(* Logix 5000 project; controller GP1 vendor 1 type 14 code 155 rev 32.11; software revision 32.01 *)
// GP1

TASK MainTask (continuous, watchdog 500 ms) : MainProgram

MODULES
   Local : vendor 1 type 14 code 155 (PointIO 0, rev 32.11)
      GP1_INPUT_MODULE_4 : 1734-IB8 (PointIO 4, rev 3.1, Input RPI 20 ms)
           Local:4:I.Data.0   // FC TOPE
           Local:4:I.Data.1   // IC TOPE
           Local:4:I.Data.3   // CAPACITIVO IZQUIERDO
           Local:4:I.Data.6   // CAPACITIVO DERECHO
      GP1_INPUT_MODULE_5 : 1734-IB8 (PointIO 5, rev 3.1, Input RPI 20 ms)
           Local:5:I.Data.0   // INDUCTIVO TOPE
           Local:5:I.Data.2   // ARRANQUE
           Local:5:I.Data.1   // PARO
           Local:5:I.Data.3   // BOTON REARME
      GP1_OUTPUT_MODULE_3 : 1734-OB8 (PointIO 3, rev 3.1, Output RPI 20 ms)
      GP1_OUTPUT_MODULE_2 : 1734-OB8 (PointIO 2, rev 3.1, Output RPI 20 ms)
           Local:2:O.Data.0   // YELLOW
           Local:2:O.Data.1   // RED
           Local:2:O.Data.2   // AZUL
      Discrete_IO : Embedded (PointIO 1, rev 32.11, Output RPI 20 ms)
           Local:1:I.Data.12   // FC CORTE SUPERIOR
           Local:1:I.Data.6   // FC CLAMP VERTICAL
           Local:1:I.Data.10   // IC CLAMP
           Local:1:I.Data.11   // FC CLAMP
           Local:1:I.Data.2   // IC NAVAJAS 3 L
           Local:1:I.Data.7   // IC CLAMP VERTICAL
           Local:1:I.Data.0   // FC NAVAJA 1
           Local:1:I.Data.1   // IC NAVAJA 1
           Local:1:I.Data.3   // FC NAVAJAS 3 L
           Local:1:I.Data.13   // IC CORTE SUPERIOR
           Local:1:I.Data.8   // IC NAVAJAS 3 R
           Local:1:I.Data.14   // IC TROQUEL
           Local:1:I.Data.15   // FC TROQUEL
           Local:1:I.Data.9   // FC NAVAJAS 3 R
           Local:1:I.Data.4   // FC CLAMP HORIZONTAL
           Local:1:I.Data.5   // IC CLAMP HORIZONTAL
           Local:1:O.Data.15   // GREEN
END_MODULES

VAR_GLOBAL   (* controller tags *)
   ACT0_OFF : BOOL := 1;   // NAVAJAS 3 R OFF
   ACT0_ON : BOOL;   // NAVAJAS 3 R ON
   ACT1_OFF : BOOL := 1;   // TROQUEL OFF
   ACT1_ON : BOOL;   // TROQUEL ON
   ACT2_OFF : BOOL := 1;   // CORTE SUPERIOR OFF
   ACT2_ON : BOOL;   // CORTE SUPERIOR ON
   ACT3_OFF : BOOL := 1;   // NAVAJA 1 OFF
   ACT3_ON : BOOL;   // NAVAJA 1 ON
   ACT4_OFF : BOOL;   // CLAMP VERTICAL OFF
   ACT4_ON : BOOL := 1;   // CLAMP VERTICAL ON
   ACT5_OFF : BOOL := 1;   // CLAMP OFF
   ACT5_ON : BOOL;   // CLAMP ON
   ACT6_OFF : BOOL;   // CLAMP HORIZONTAL OFF
   ACT6_ON : BOOL := 1;   // CLAMP HORIZONTAL ON
   ACT7_OFF : BOOL := 1;   // NAVAJA 3 L OFF
   ACT7_ON : BOOL;   // NAVAJA 3 L ON
   ACT8_OFF : BOOL;   // TOPE OFF
   ACT8_ON : BOOL := 1;   // TOPE ON
   AIR_ALARM : BOOL;
   ALARM_TIM : TIMER := (PRE := 5000);
   ALARMED : BOOL;
   ARRANQUE_AUTO : BOOL;
   AUTO : BOOL;
   C1 : COUNTER := (ACC := 5, DN := 1);
   CAPACITIVE_SENSOR_1 : BOOL;
   CAPACITIVE_SENSOR_2 : BOOL;
   CND1 : BOOL;
   CND10 : BOOL;
   CND2 : BOOL;
   CND3 : BOOL;
   CND4 : BOOL;
   CND5 : BOOL;
   CND6 : BOOL;
   CND7 : BOOL;
   CND8 : BOOL;
   CND9 : BOOL;
   CORTE_VALVULA : BOOL;
   CORTINA_SEG : BOOL := 1;
   CT : COUNTER := (ACC := 47, DN := 1);
   CURRENT_SCREEN : DINT;
   E_STOP : BOOL;
   E_STOP_ALARM : BOOL;
   EstadoHMI : DINT := 2;
   EVBI0_AUTO_OFF : BOOL;   // NAVAJAS 3 OFF AUTO
   EVBI0_AUTO_ON : BOOL;   // NAVAJAS 3 ON AUTO
   EVBI0_MAN_OFF : BOOL;   // NAVAJAS 3 OFF MANUAL
   EVBI0_MAN_ON : BOOL;   // NAVAJAS 3 ON MANUAL
   EVBI0_OFF : BOOL := 1;   // NAVAJAS 3 OFF
   EVBI0_ON : BOOL;   // NAVAJAS 3 ON
   EVBI1_AUTO_OFF : BOOL;   // TROQUEL OFF AUTO
   EVBI1_AUTO_ON : BOOL;   // TROQUEL ON AUTO
   EVBI1_MAN_OFF : BOOL;   // TROQUEL OFF MANUAL
   EVBI1_MAN_ON : BOOL;   // TROQUEL ON MANUAL
   EVBI1_OFF : BOOL := 1;   // TROQUEL OFF
   EVBI1_ON : BOOL;   // TROQUEL ON
   EVBI2_AUTO_OFF : BOOL;   // CLAMP OFF AUTO
   EVBI2_AUTO_ON : BOOL;   // CLAMP ON AUTO
   EVBI2_MAN_OFF : BOOL;   // CLAMP OFF MANUAL
   EVBI2_MAN_ON : BOOL;   // CLAMP ON MANUAL
   EVBI2_OFF : BOOL := 1;   // CLAMP OFF
   EVBI2_ON : BOOL;   // CLAMP ON
   EVBI3_AUTO_OFF : BOOL;   // NAVAJA 1 OFF AUTO
   EVBI3_AUTO_ON : BOOL;   // NAVAJA 1 ON AUTO
   EVBI3_MAN_OFF : BOOL;   // NAVAJA 1 OFF MANUAL
   EVBI3_MAN_ON : BOOL;   // NAVAJA 1 ON MANUAL
   EVBI3_OFF : BOOL := 1;   // NAVAJA 1 OFF
   EVBI3_ON : BOOL;   // NAVAJA 1 ON
   EVBI4_AUTO_OFF : BOOL;   // CLAMP VERTICAL OFF AUTO
   EVBI4_AUTO_ON : BOOL;   // CLAMP VERTICAL ON AUTO
   EVBI4_MAN_OFF : BOOL;   // CLAMP VERTICAL OFF MANUAL
   EVBI4_MAN_ON : BOOL;   // CLAMP VERTICAL ON MANUAL
   EVBI4_OFF : BOOL;   // CLAMP VERTICAL OFF
   EVBI4_ON : BOOL := 1;   // CLAMP VERTICAL ON
   EVBI5_AUTO_OFF : BOOL;   // CORTE SUPERIOR OFF AUTO
   EVBI5_AUTO_ON : BOOL;   // CORTE SUPERIOR ON AUTO
   EVBI5_MAN_OFF : BOOL;   // CORTE SUPERIOR OFF MANUAL
   EVBI5_MAN_ON : BOOL;   // CORTE SUPERIOR ON MANUAL
   EVBI5_OFF : BOOL := 1;   // CORTE SUPERIOR OFF
   EVBI5_ON : BOOL;   // CORTE SUPERIOR ON
   EVBI6_AUTO_OFF : BOOL;   // CLAMP HORIZONTAL OFF AUTO
   EVBI6_AUTO_ON : BOOL;   // CLAMP HORIZONTAL ON AUTO
   EVBI6_MAN_OFF : BOOL;   // CLAMP HORIZONTAL OFF MANUAL
   EVBI6_MAN_ON : BOOL;   // CLAMP HORIZONTAL ON MANUAL
   EVBI6_OFF : BOOL;   // CLAMP HORIZONTAL OFF
   EVBI6_ON : BOOL := 1;   // CLAMP HORIZONTAL ON
   EVMONO1_AUTO_OFF : BOOL;
   EVMONO1_AUTO_ON : BOOL;   // TOPE_AUTO_ON
   EVMONO1_MAN_OFF : BOOL;
   EVMONO1_MAN_ON : BOOL;
   EVMONO_OFF : BOOL;
   EVMONO_ON : BOOL;   // TOPE ON
   EXCEDDED_TIME_FOR_CILINDERS : BOOL;
   EXCEDDED_TIME_FOR_INIT_COND : BOOL;
   FAIL_COUNT : COUNTER;
   GREEN_LIGHT : BOOL;
   INITIAL_CONDITIONS_NOT_READY : BOOL := 1;
   INITIAL_CONDITIONS_READY : BOOL;
   L_S_OK : BOOL := 1;   // SENSOR IZQUIERDO
   LAMP : BOOL := 1;
   LATCH_TEST : BOOL;
   LIGHT_CURTAIN : BOOL;
   MAN_SCREENS : BOOL;   // PANTALLAS MANUALES
   MANUAL : BOOL := 1;
   MSJ_CND_INIT : DINT := 8;
   NO_AIR : BOOL;
   NO_ALARM : BOOL := 1;
   NOT_CORRECTLY_PLACED : BOOL;
   OBESTOP : BOOL;
   OK : BOOL;
   ONS1 : BOOL;
   PARO : BOOL := 1;
   Paso1 : BOOL;
   Paso10 : BOOL;
   Paso11 : BOOL;
   Paso12 : BOOL;
   Paso13 : BOOL;
   Paso14 : BOOL;
   Paso15 : BOOL;
   Paso16 : BOOL;
   Paso17 : BOOL;
   Paso18 : BOOL;
   Paso2 : BOOL;
   Paso3 : BOOL;
   Paso4 : BOOL;
   Paso5 : BOOL;
   Paso6 : BOOL;
   Paso7 : BOOL;
   Paso8 : BOOL;
   Paso9 : BOOL;
   Paso_Sec : DINT;
   PIECE_PLACED : BOOL;
   PRESOSTATO : BOOL := 1;
   R_S_OK : BOOL := 1;   // SENSOR DERECHO
   REARME_OK : BOOL;
   REARMY_BUTTON : BOOL;
   REARMY_TIME : TIMER := (PRE := 5);
   REARMY_WARNING : BOOL := 1;   // LUZ DE ARME
   RED_LIGHT : BOOL;
   REPEATED_ALARM : BOOL;
   RESET_COUNTER : BOOL;
   RESET_LATCH_TEST : BOOL;
   SAFETY_CURTAIN : BOOL;
   SAFETY_CURTAIN_ALARM : BOOL;
   SBESTOP : BOOL;
   SENSOR1 : BOOL;
   SENSOR_TOPE : BOOL;   // TOPE DE PIEZA
   Sequence_ON : BOOL;
   Start_Sequence : BOOL;
   T1 : TIMER := (PRE := 300);
   T10 : TIMER := (PRE := 300);
   T11 : TIMER := (PRE := 300);
   T12 : TIMER := (PRE := 300);
   T13 : TIMER := (PRE := 300);
   T14 : TIMER := (PRE := 300);
   T15 : TIMER := (PRE := 300);
   T16 : TIMER := (PRE := 300);
   T17 : TIMER := (PRE := 300);
   T18 : TIMER := (PRE := 1000);
   T2 : TIMER := (PRE := 300);
   T3 : TIMER := (PRE := 300);
   T4 : TIMER := (PRE := 300);
   T5 : TIMER := (PRE := 300);
   T6 : TIMER := (PRE := 300);
   T7 : TIMER := (PRE := 300);
   T8 : TIMER := (PRE := 300);
   T9 : TIMER := (PRE := 300);
   TCLAMP : TIMER := (PRE := 250, ACC := 250, EN := 1, DN := 1);
   TEST : BOOL;
   TEST_2 : BOOL;
   TEST_3 : BOOL;
   TEST_RESET : BOOL;
   TEST_STOP : BOOL;
   TIMOFF : TIMER := (PRE := 500);
   TIMON : TIMER := (PRE := 500);
   TIMSACC : DINT;
   TIMW1 : TIMER := (PRE := 2000);
   TIMW2 : TIMER := (PRE := 1);
   USER : DINT;
   WAITING : BOOL;
   WORKING : BOOL;
   YELLOW_LIGHT : BOOL := 1;
END_VAR

PROGRAM MainProgram   (* main routine MainRoutine *)
VAR
   BYPASS_DER : BOOL;
   BYPASS_IZQ : BOOL;
   BYPASS_TOPE : BOOL;
   BypassStatus : DINT;
   CERRARSESION : BOOL;
   ING_ACCESS : BOOL;
   LOGOUT : BOOL;
   MTTO_ACCESS : BOOL;
   RESET_COUNTERT : BOOL;
   TEMP1 : BOOL;
   TEMP2 : BOOL;
   TEMP3 : BOOL;
   USERstring : STRING;
END_VAR

ROUTINE ALARMS   (* ladder *)
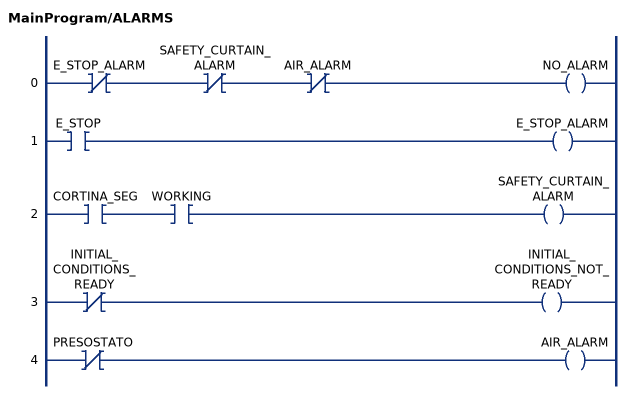
   0: XIO(E_STOP_ALARM)XIO(SAFETY_CURTAIN_ALARM)XIO(AIR_ALARM)OTE(NO_ALARM);
   1: XIC(E_STOP)OTE(E_STOP_ALARM);
   2: XIC(CORTINA_SEG)XIC(WORKING)OTE(SAFETY_CURTAIN_ALARM);
   3: XIO(INITIAL_CONDITIONS_READY)OTE(INITIAL_CONDITIONS_NOT_READY);
   4: XIO(PRESOSTATO)OTE(AIR_ALARM);
END_ROUTINE

ROUTINE AUTO_SEQUENCE   (* ladder *)
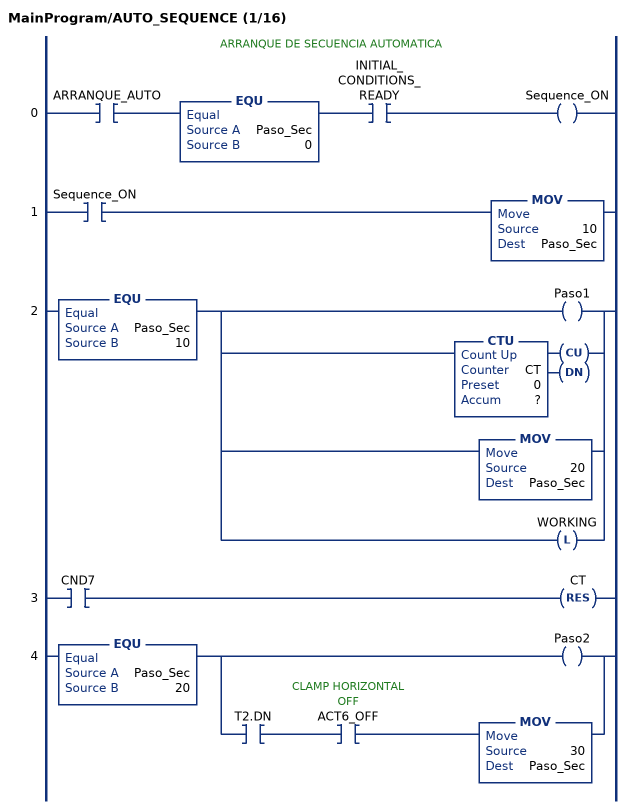
   // ARRANQUE DE SECUENCIA AUTOMATICA
   0: XIC(ARRANQUE_AUTO)EQU(Paso_Sec,0)XIC(INITIAL_CONDITIONS_READY)OTE(Sequence_ON);
   1: XIC(Sequence_ON)MOV(10,Paso_Sec);
   2: EQU(Paso_Sec,10)[OTE(Paso1) ,CTU(CT,?,?) ,MOV(20,Paso_Sec) ,OTL(WORKING) ];
   3: XIC(CND7)RES(CT);
   4: EQU(Paso_Sec,20)[OTE(Paso2) ,XIC(T2.DN) XIC(ACT6_OFF) MOV(30,Paso_Sec) ];
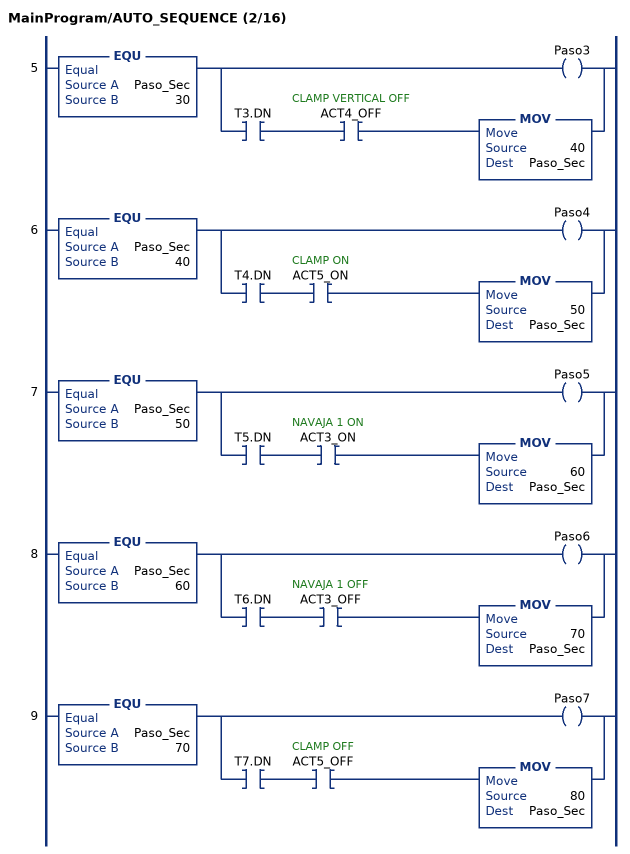
   5: EQU(Paso_Sec,30)[OTE(Paso3) ,XIC(T3.DN) XIC(ACT4_OFF) MOV(40,Paso_Sec) ];
   6: EQU(Paso_Sec,40)[OTE(Paso4) ,XIC(T4.DN) XIC(ACT5_ON) MOV(50,Paso_Sec) ];
   7: EQU(Paso_Sec,50)[OTE(Paso5) ,XIC(T5.DN) XIC(ACT3_ON) MOV(60,Paso_Sec) ];
   8: EQU(Paso_Sec,60)[OTE(Paso6) ,XIC(T6.DN) XIC(ACT3_OFF) MOV(70,Paso_Sec) ];
   9: EQU(Paso_Sec,70)[OTE(Paso7) ,XIC(T7.DN) XIC(ACT5_OFF) MOV(80,Paso_Sec) ];
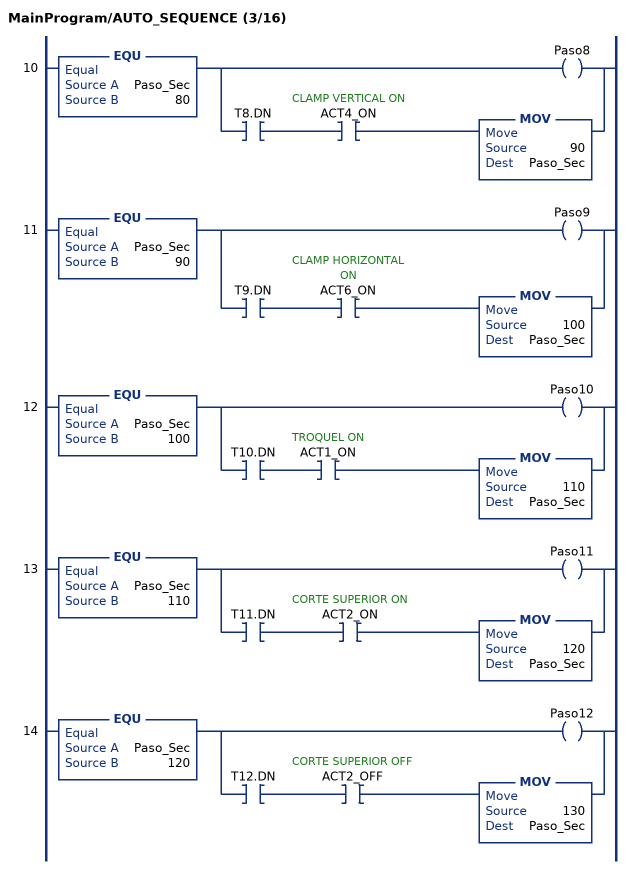
   10: EQU(Paso_Sec,80)[OTE(Paso8) ,XIC(T8.DN) XIC(ACT4_ON) MOV(90,Paso_Sec) ];
   11: EQU(Paso_Sec,90)[OTE(Paso9) ,XIC(T9.DN) XIC(ACT6_ON) MOV(100,Paso_Sec) ];
   12: EQU(Paso_Sec,100)[OTE(Paso10) ,XIC(T10.DN) XIC(ACT1_ON) MOV(110,Paso_Sec) ];
   13: EQU(Paso_Sec,110)[OTE(Paso11) ,XIC(T11.DN) XIC(ACT2_ON) MOV(120,Paso_Sec) ];
   14: EQU(Paso_Sec,120)[OTE(Paso12) ,XIC(T12.DN) XIC(ACT2_OFF) MOV(130,Paso_Sec) ];
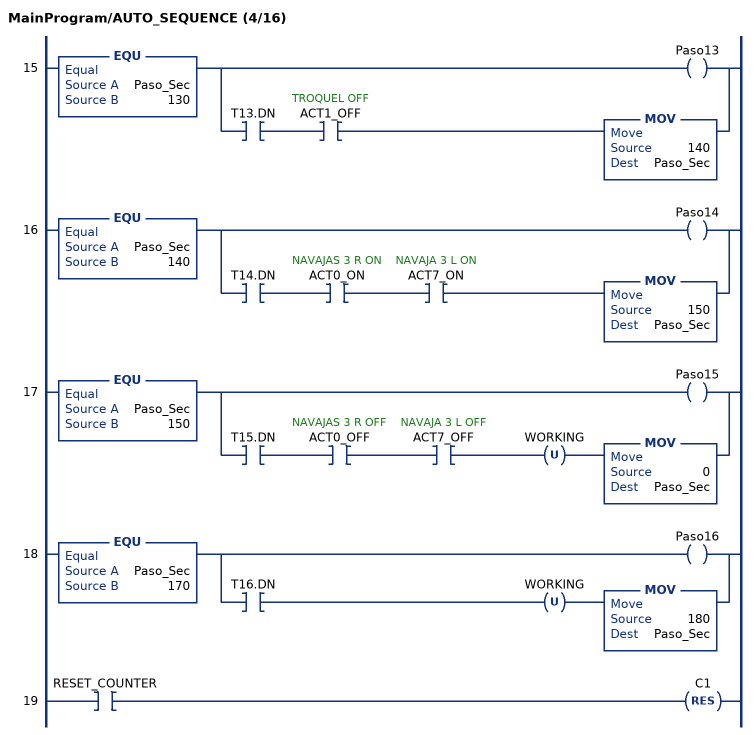
   15: EQU(Paso_Sec,130)[OTE(Paso13) ,XIC(T13.DN) XIC(ACT1_OFF) MOV(140,Paso_Sec) ];
   16: EQU(Paso_Sec,140)[OTE(Paso14) ,XIC(T14.DN) XIC(ACT0_ON) XIC(ACT7_ON) MOV(150,Paso_Sec) ];
   17: EQU(Paso_Sec,150)[OTE(Paso15) ,XIC(T15.DN) XIC(ACT0_OFF) XIC(ACT7_OFF) OTU(WORKING) MOV(0,Paso_Sec) ];
   18: EQU(Paso_Sec,170)[OTE(Paso16) ,XIC(T16.DN) OTU(WORKING) MOV(180,Paso_Sec) ];
   19: XIC(RESET_COUNTER)RES(C1);
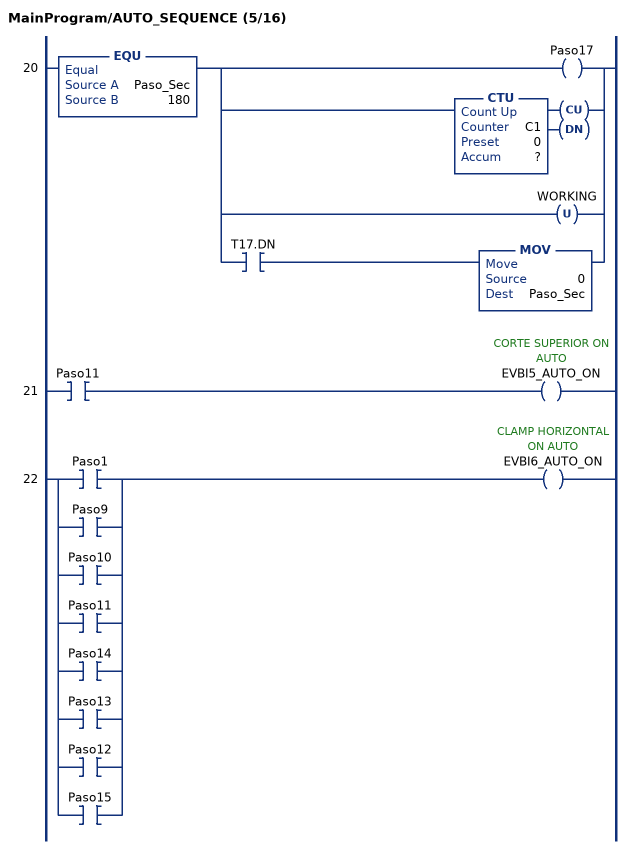
   20: EQU(Paso_Sec,180)[OTE(Paso17) ,CTU(C1,?,?) ,OTU(WORKING) ,XIC(T17.DN) MOV(0,Paso_Sec) ];
   21: XIC(Paso11)OTE(EVBI5_AUTO_ON);
   22: [XIC(Paso1) ,XIC(Paso9) ,XIC(Paso10) ,XIC(Paso11) ,XIC(Paso14) ,XIC(Paso13) ,XIC(Paso12) ,XIC(Paso15) ]OTE(EVBI6_AUTO_ON);
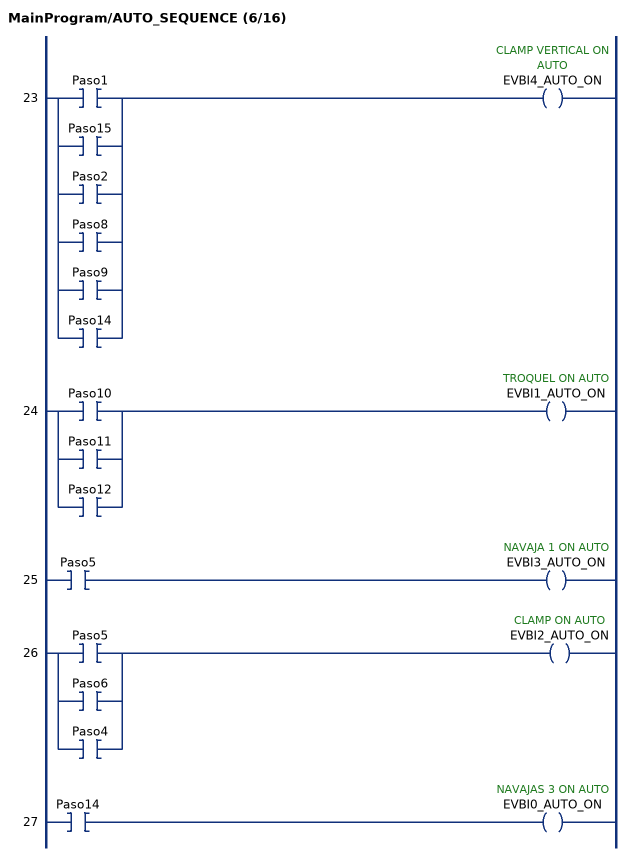
   23: [XIC(Paso1) ,XIC(Paso15) ,XIC(Paso2) ,XIC(Paso8) ,XIC(Paso9) ,XIC(Paso14) ]OTE(EVBI4_AUTO_ON);
   24: [XIC(Paso10) ,XIC(Paso11) ,XIC(Paso12) ]OTE(EVBI1_AUTO_ON);
   25: XIC(Paso5)OTE(EVBI3_AUTO_ON);
   26: [XIC(Paso5) ,XIC(Paso6) ,XIC(Paso4) ]OTE(EVBI2_AUTO_ON);
   27: XIC(Paso14)OTE(EVBI0_AUTO_ON);
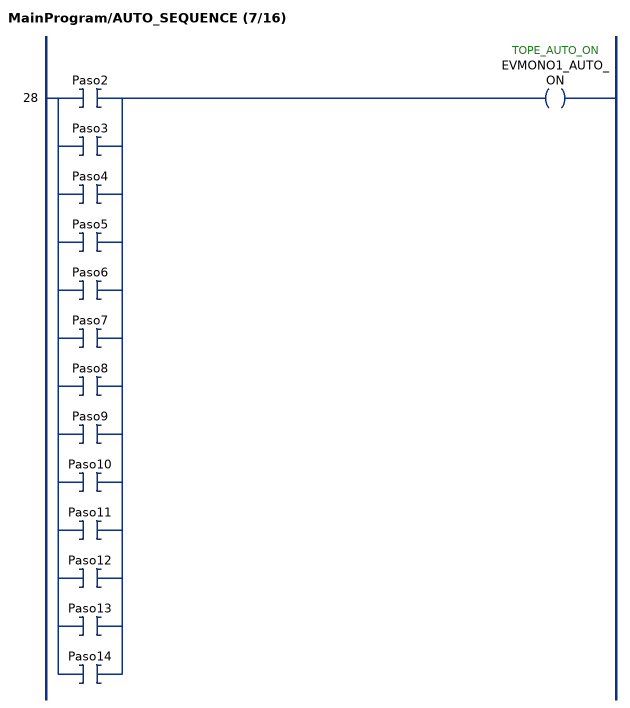
   28: [XIC(Paso2) ,XIC(Paso3) ,XIC(Paso4) ,XIC(Paso5) ,XIC(Paso6) ,XIC(Paso7) ,XIC(Paso8) ,XIC(Paso9) ,XIC(Paso10) ,XIC(Paso11) ,XIC(Paso12) ,XIC(Paso13) ,XIC(Paso14) ]OTE(EVMONO1_AUTO_ON);
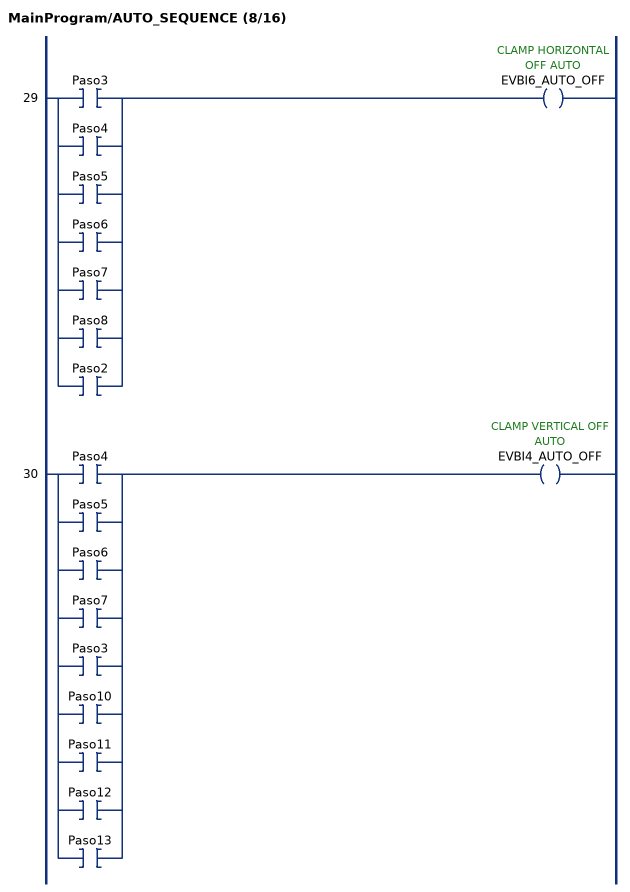
   29: [XIC(Paso3) ,XIC(Paso4) ,XIC(Paso5) ,XIC(Paso6) ,XIC(Paso7) ,XIC(Paso8) ,XIC(Paso2) ]OTE(EVBI6_AUTO_OFF);
   30: [XIC(Paso4) ,XIC(Paso5) ,XIC(Paso6) ,XIC(Paso7) ,XIC(Paso3) ,XIC(Paso10) ,XIC(Paso11) ,XIC(Paso12) ,XIC(Paso13) ]OTE(EVBI4_AUTO_OFF);
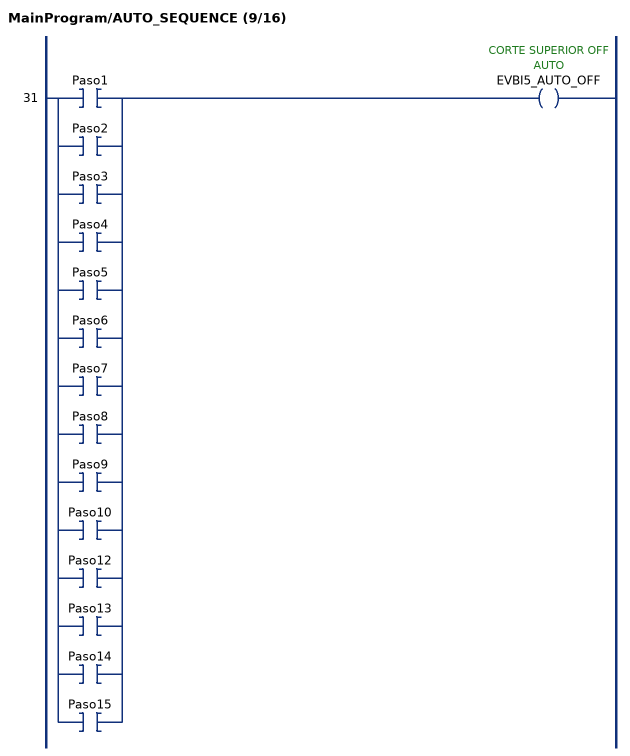
   31: [XIC(Paso1) ,XIC(Paso2) ,XIC(Paso3) ,XIC(Paso4) ,XIC(Paso5) ,XIC(Paso6) ,XIC(Paso7) ,XIC(Paso8) ,XIC(Paso9) ,XIC(Paso10) ,XIC(Paso12) ,XIC(Paso13) ,XIC(Paso14) ,XIC(Paso15) ]OTE(EVBI5_AUTO_OFF);
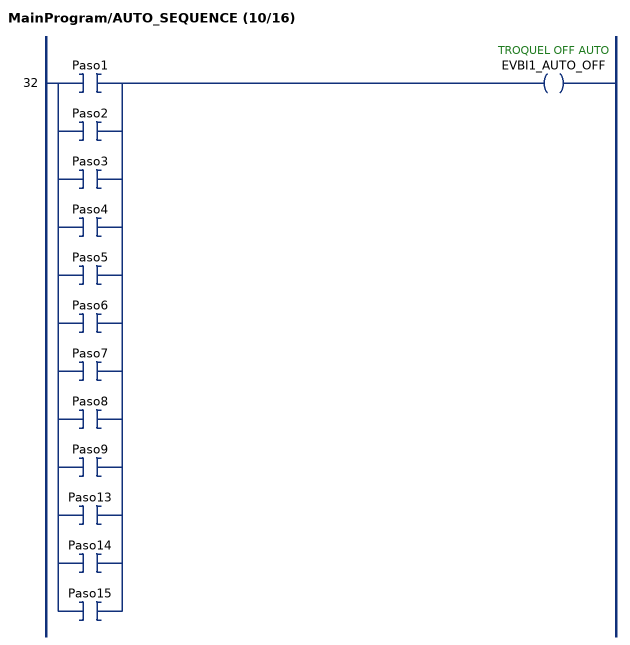
   32: [XIC(Paso1) ,XIC(Paso2) ,XIC(Paso3) ,XIC(Paso4) ,XIC(Paso5) ,XIC(Paso6) ,XIC(Paso7) ,XIC(Paso8) ,XIC(Paso9) ,XIC(Paso13) ,XIC(Paso14) ,XIC(Paso15) ]OTE(EVBI1_AUTO_OFF);
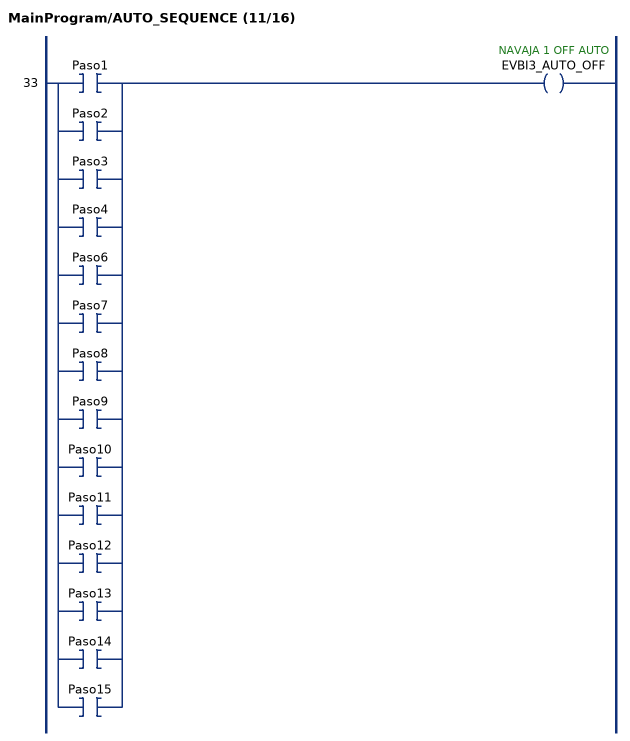
   33: [XIC(Paso1) ,XIC(Paso2) ,XIC(Paso3) ,XIC(Paso4) ,XIC(Paso6) ,XIC(Paso7) ,XIC(Paso8) ,XIC(Paso9) ,XIC(Paso10) ,XIC(Paso11) ,XIC(Paso12) ,XIC(Paso13) ,XIC(Paso14) ,XIC(Paso15) ]OTE(EVBI3_AUTO_OFF);
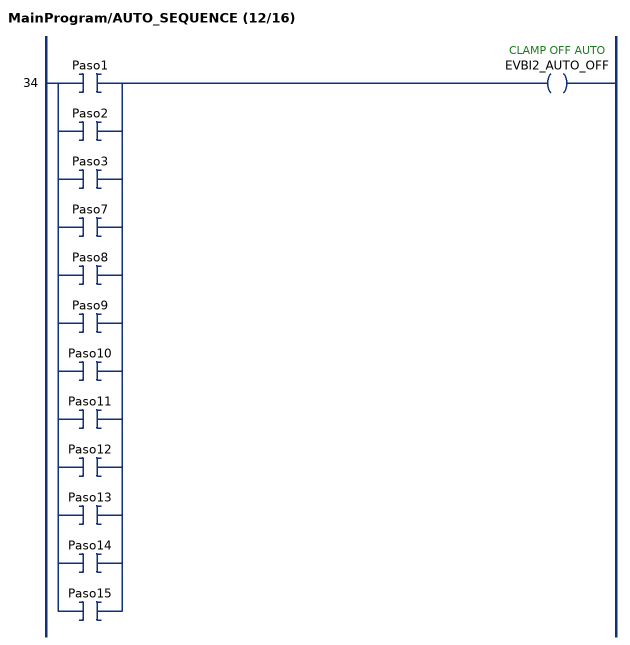
   34: [XIC(Paso1) ,XIC(Paso2) ,XIC(Paso3) ,XIC(Paso7) ,XIC(Paso8) ,XIC(Paso9) ,XIC(Paso10) ,XIC(Paso11) ,XIC(Paso12) ,XIC(Paso13) ,XIC(Paso14) ,XIC(Paso15) ]OTE(EVBI2_AUTO_OFF);
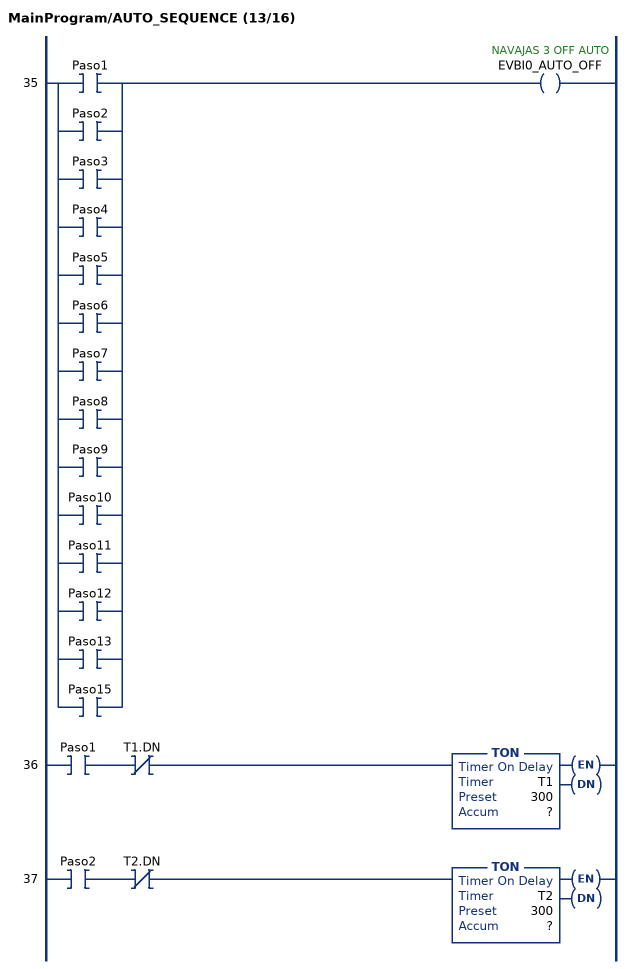
   35: [XIC(Paso1) ,XIC(Paso2) ,XIC(Paso3) ,XIC(Paso4) ,XIC(Paso5) ,XIC(Paso6) ,XIC(Paso7) ,XIC(Paso8) ,XIC(Paso9) ,XIC(Paso10) ,XIC(Paso11) ,XIC(Paso12) ,XIC(Paso13) ,XIC(Paso15) ]OTE(EVBI0_AUTO_OFF);
   36: XIC(Paso1)XIO(T1.DN)TON(T1,?,?);
   37: XIC(Paso2)XIO(T2.DN)TON(T2,?,?);
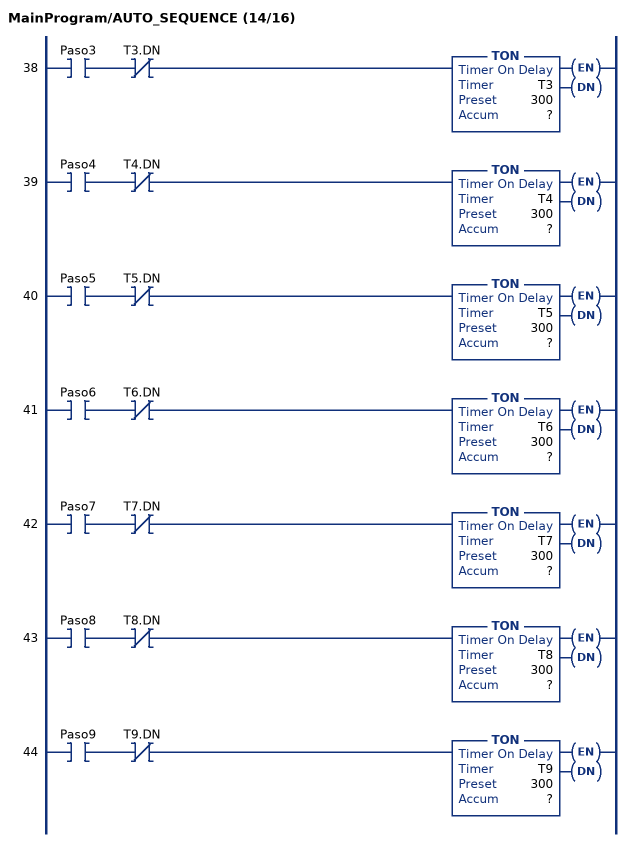
   38: XIC(Paso3)XIO(T3.DN)TON(T3,?,?);
   39: XIC(Paso4)XIO(T4.DN)TON(T4,?,?);
   40: XIC(Paso5)XIO(T5.DN)TON(T5,?,?);
   41: XIC(Paso6)XIO(T6.DN)TON(T6,?,?);
   42: XIC(Paso7)XIO(T7.DN)TON(T7,?,?);
   43: XIC(Paso8)XIO(T8.DN)TON(T8,?,?);
   44: XIC(Paso9)XIO(T9.DN)TON(T9,?,?);
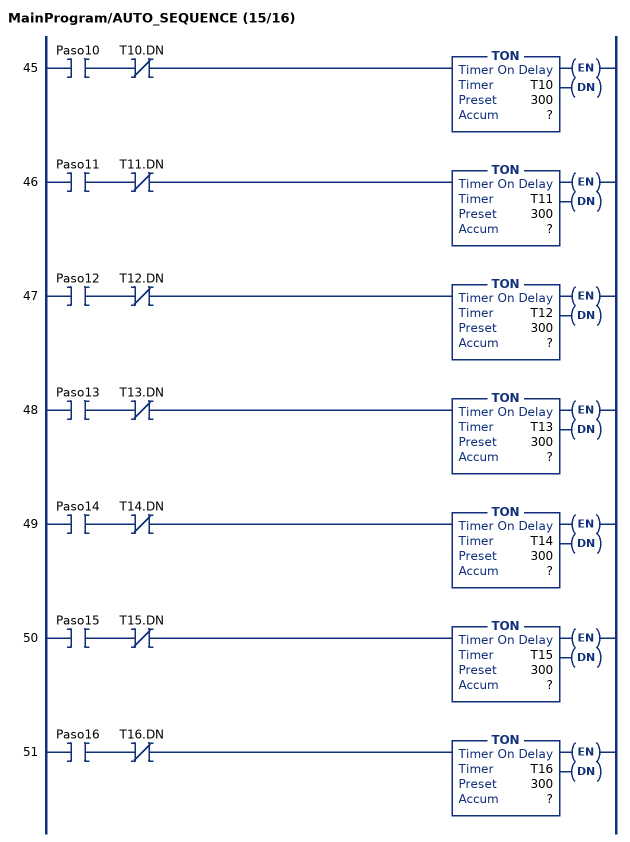
   45: XIC(Paso10)XIO(T10.DN)TON(T10,?,?);
   46: XIC(Paso11)XIO(T11.DN)TON(T11,?,?);
   47: XIC(Paso12)XIO(T12.DN)TON(T12,?,?);
   48: XIC(Paso13)XIO(T13.DN)TON(T13,?,?);
   49: XIC(Paso14)XIO(T14.DN)TON(T14,?,?);
   50: XIC(Paso15)XIO(T15.DN)TON(T15,?,?);
   51: XIC(Paso16)XIO(T16.DN)TON(T16,?,?);
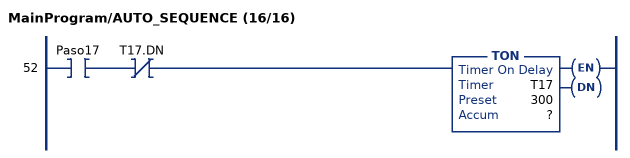
   52: XIC(Paso17)XIO(T17.DN)TON(T17,?,?);
END_ROUTINE

ROUTINE INPUTS   (* ladder *)
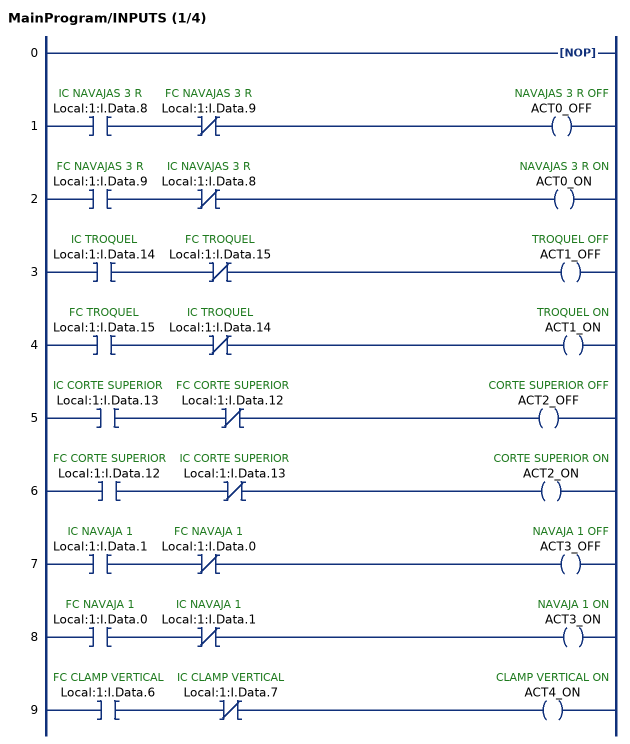
   0: NOP();
   1: XIC(Local:1:I.Data.8)XIO(Local:1:I.Data.9)OTE(ACT0_OFF);
   2: XIC(Local:1:I.Data.9)XIO(Local:1:I.Data.8)OTE(ACT0_ON);
   3: XIC(Local:1:I.Data.14)XIO(Local:1:I.Data.15)OTE(ACT1_OFF);
   4: XIC(Local:1:I.Data.15)XIO(Local:1:I.Data.14)OTE(ACT1_ON);
   5: XIC(Local:1:I.Data.13)XIO(Local:1:I.Data.12)OTE(ACT2_OFF);
   6: XIC(Local:1:I.Data.12)XIO(Local:1:I.Data.13)OTE(ACT2_ON);
   7: XIC(Local:1:I.Data.1)XIO(Local:1:I.Data.0)OTE(ACT3_OFF);
   8: XIC(Local:1:I.Data.0)XIO(Local:1:I.Data.1)OTE(ACT3_ON);
   9: XIC(Local:1:I.Data.6)XIO(Local:1:I.Data.7)OTE(ACT4_ON);
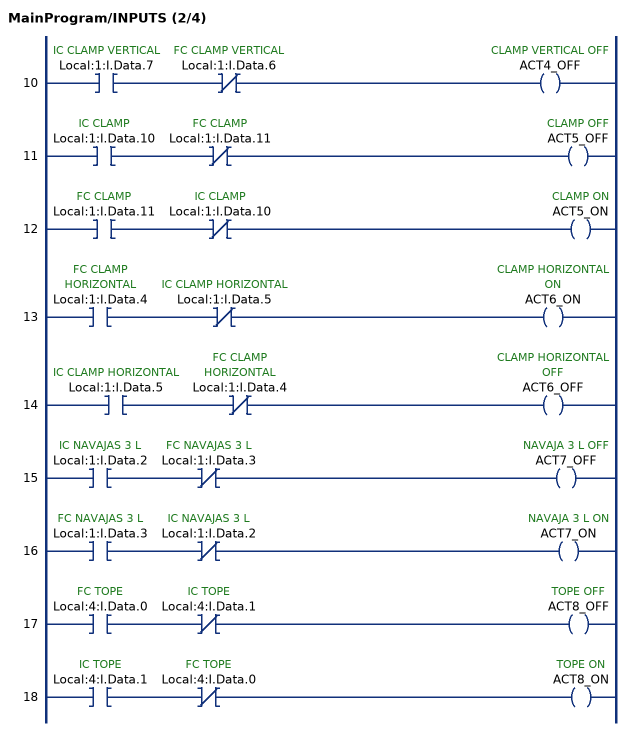
   10: XIC(Local:1:I.Data.7)XIO(Local:1:I.Data.6)OTE(ACT4_OFF);
   11: XIC(Local:1:I.Data.10)XIO(Local:1:I.Data.11)OTE(ACT5_OFF);
   12: XIC(Local:1:I.Data.11)XIO(Local:1:I.Data.10)OTE(ACT5_ON);
   13: XIC(Local:1:I.Data.4)XIO(Local:1:I.Data.5)OTE(ACT6_ON);
   14: XIC(Local:1:I.Data.5)XIO(Local:1:I.Data.4)OTE(ACT6_OFF);
   15: XIC(Local:1:I.Data.2)XIO(Local:1:I.Data.3)OTE(ACT7_OFF);
   16: XIC(Local:1:I.Data.3)XIO(Local:1:I.Data.2)OTE(ACT7_ON);
   17: XIC(Local:4:I.Data.0)XIO(Local:4:I.Data.1)OTE(ACT8_OFF);
   18: XIC(Local:4:I.Data.1)XIO(Local:4:I.Data.0)OTE(ACT8_ON);
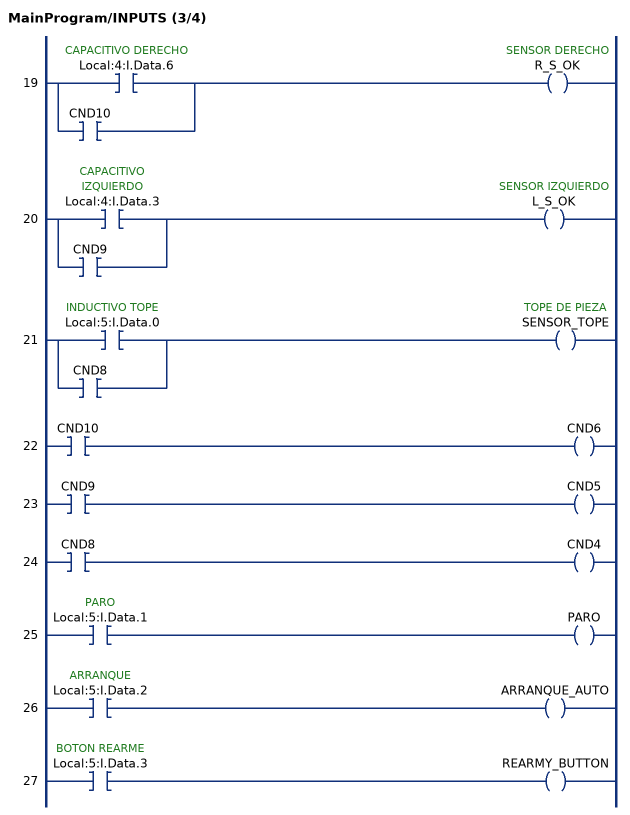
   19: [XIC(Local:4:I.Data.6) ,XIC(CND10) ]OTE(R_S_OK);
   20: [XIC(Local:4:I.Data.3) ,XIC(CND9) ]OTE(L_S_OK);
   21: [XIC(Local:5:I.Data.0) ,XIC(CND8) ]OTE(SENSOR_TOPE);
   22: XIC(CND10)OTE(CND6);
   23: XIC(CND9)OTE(CND5);
   24: XIC(CND8)OTE(CND4);
   25: XIC(Local:5:I.Data.1)OTE(PARO);
   26: XIC(Local:5:I.Data.2)OTE(ARRANQUE_AUTO);
   27: XIC(Local:5:I.Data.3)OTE(REARMY_BUTTON);
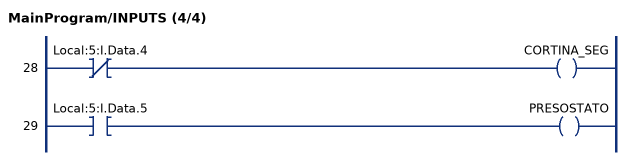
   28: XIO(Local:5:I.Data.4)OTE(CORTINA_SEG);
   29: XIC(Local:5:I.Data.5)OTE(PRESOSTATO);
END_ROUTINE
